PROGRAM MAIN
VAR
	fbWritePersistentData	: FB_WritePersistentData; (* Chamada do bloco para salvar variáveis persistentes*)
	fbClock					: FB_CLOCK; (* Bloco CLOCK *)
END_VAR

ACT_Persistent(); (* Action com os blocos persistentes *)

P_LubLogic(); (* Lógica de Lubrificação *)

ACTION ACT_Persistent:
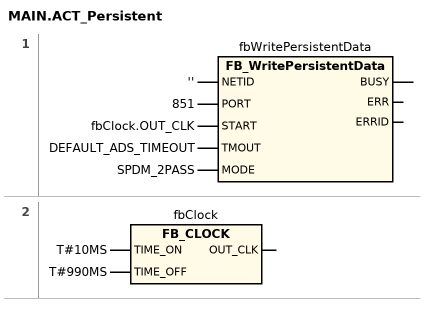
// NETWORK 1
fbWritePersistentData(
    NETID := '',
    PORT := 851,
    START := fbClock.OUT_CLK,
    TMOUT := DEFAULT_ADS_TIMEOUT,
    MODE := SPDM_2PASS); // FB_WritePersistentData

// NETWORK 2
fbClock(TIME_ON := T#10MS, TIME_OFF := T#990MS); // FB_CLOCK
END_ACTION

END_PROGRAM

(* stored: Version 1.1.0.1, ProductVersion 3.1.4024.12
   POU MAIN: Id {9f9d47eb-c6d0-4cee-b565-0572ddc430ba}, SpecialFunc None
   Action ACT_Persistent: Id {5fa1b91a-99a2-4c3f-9850-c3b3d13b553d} *)
